// TIA Portal V20 export
ORGANIZATION_BLOCK "CFC_Startup"   // OB1100, CFC, Startup
TITLE = "Complete Restart"
{ S7_Optimized_Access := 'TRUE' }
AUTHOR : CFC
FAMILY : CFCPlus
VERSION : 1.0
// stored: AutoNumber false
   VAR_INPUT
      LostRetentive : Bool;   // True if retentive data are lost
      LostRTC : Bool;   // True if date and time are lost
   END_VAR
   VAR_TEMP
      t_out : UInt;
   END_VAR
BEGIN
END_ORGANIZATION_BLOCK
